// TIA Portal project "Encoder_Ve_Hızlı_Sayıcı_Uygulaması_V1" (V16)

(* hardware
DEVICE "S7-1200 station_1"  S7-1200 Station
   slot 0: "Rack_0"  S7-1200 Rack  Rack  V1.0
   slot 1: "PLC_1"  CPU 1214C DC/DC/DC  6ES7 214-1AG40-0XB0  V4.4
*)

// ===== PLC "PLC_1"  CPU 1214C DC/DC/DC =====

VAR_GLOBAL   // PLC tag table "Default tag table"
   "Tag_1" AT %ID1000 : DInt;
   "Tur_Sayısı" AT %MD20 : DInt;
   "Çıkış_1" AT %Q0.0 : Bool;
   "Tag_2" AT %M10.0 : Bool;
END_VAR

ORGANIZATION_BLOCK "Main"   // OB1, LAD, ProgramCycle
TITLE = "Main Program Sweep (Cycle)"
{ S7_Optimized_Access := 'TRUE' }
VERSION : 0.1
   VAR_INPUT
      Initial_Call : Bool;   // Initial call of this OB
      Remanence : Bool;   // =True, if remanent data are available
   END_VAR
BEGIN

REGION Network 1: Motorun Tur Sayısını Hesaplama
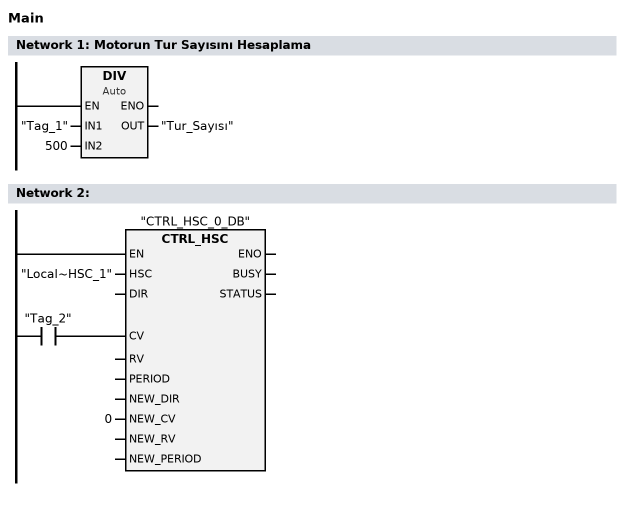
   RUNG wire#powerrail
      Div(in1 := "Tag_1", in2 := 500, out => "Tur_Sayısı")
   END_RUNG
   // the same network as SCL:
   "Tur_Sayısı" := "Tag_1" / 500;
END_REGION

REGION Network 2
   "CTRL_HSC_0_DB"(HSC := "Local~HSC_1", CV := "Tag_2", NEW_CV := 0);   // CTRL_HSC
END_REGION
END_ORGANIZATION_BLOCK

ORGANIZATION_BLOCK "Hardware interrupt"   // OB40, LAD, HWProcessInterrupt
{ S7_Optimized_Access := 'TRUE' }
VERSION : 0.1
   VAR_INPUT
      LADDR : Hw_Io;   // Hardware identifier
      USI : Word;   // User structure identifier
      IChannel : USInt;   // Interrupt channel number
      EventType : Byte;   // EventType
   END_VAR
BEGIN

REGION Network 1: Kesme oluştuğunda çıkışları aktif etme
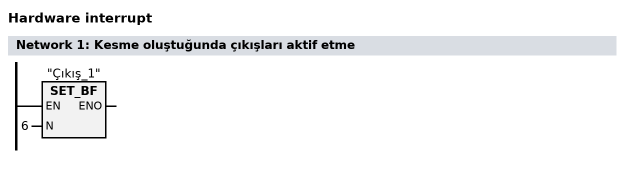
   // no SCL statement known for SBitfield: written as a call
   SET_BF(operand := "Çıkış_1", n := 6);
END_REGION
END_ORGANIZATION_BLOCK